FUNCTION_BLOCK FB_Mixer_Ctrl
VAR_INPUT
	i_Interlocks		:ARRAY[1..5] OF BOOL;
	i_AutoCmdFwd		:BOOL;
	i_AutoCmdBcw		:BOOL;
	i_AutoSpeedSP		:REAL;
	i_ManCmdFwd			:BOOL;
	i_ManCmdBcw			:BOOL;
	i_ManStop			:BOOL;
	i_ManSpeedSP		:REAL;
	i_SpeedAP			:REAL;
	i_CurrentAP			:REAL;
	i_ServiceMode		:BOOL;
END_VAR
VAR_OUTPUT
	q_InterlocksOK		:BOOL;
	q_bCmdFwd			:BOOL;
	q_bCmdBcw			:BOOL;
	q_rSpeedSP			:REAL;
END_VAR
VAR
	bCmdFwd				:BOOL;
	bCmdBcw				:BOOL;
	tofCMDFwd			:TOF;
	tofCMDBcw			:TOF;
	tonFwdOff			:TON;
	tonBcwOff			:TON;
END_VAR
VAR // added by the converter: edge detectors and wires of the graphical bodies
    _w1 : BOOL;
END_VAR

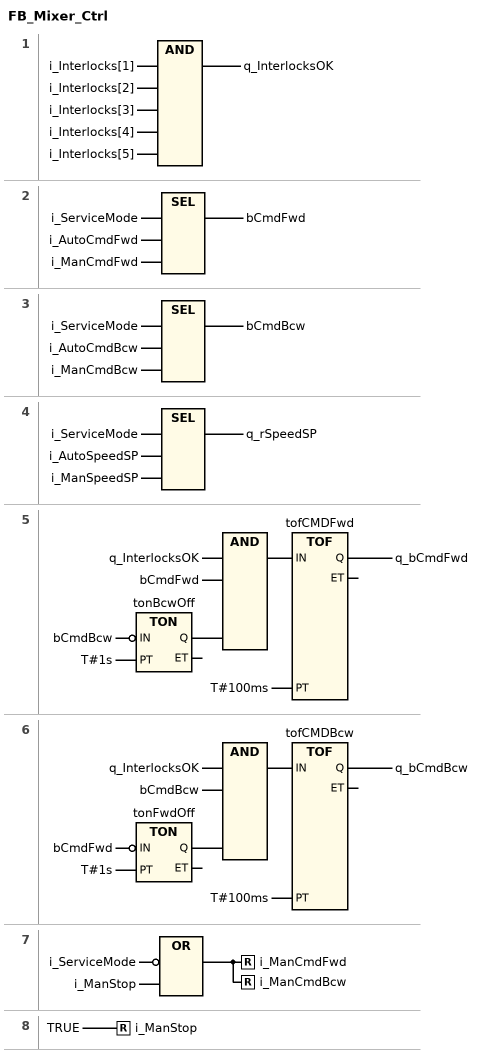
// NETWORK 1
q_InterlocksOK := i_Interlocks[1] AND i_Interlocks[2] AND i_Interlocks[3] AND i_Interlocks[4] AND i_Interlocks[5];

// NETWORK 2
bCmdFwd := SEL(i_ServiceMode, i_AutoCmdFwd, i_ManCmdFwd);

// NETWORK 3
bCmdBcw := SEL(i_ServiceMode, i_AutoCmdBcw, i_ManCmdBcw);

// NETWORK 4
q_rSpeedSP := SEL(i_ServiceMode, i_AutoSpeedSP, i_ManSpeedSP);

// NETWORK 5
tonBcwOff(IN := NOT bCmdBcw, PT := T#1s); // TON
tofCMDFwd(IN := q_InterlocksOK AND bCmdFwd AND tonBcwOff.Q, PT := T#100ms); // TOF
q_bCmdFwd := tofCMDFwd.Q;

// NETWORK 6
tonFwdOff(IN := NOT bCmdFwd, PT := T#1s); // TON
tofCMDBcw(IN := q_InterlocksOK AND bCmdBcw AND tonFwdOff.Q, PT := T#100ms); // TOF
q_bCmdBcw := tofCMDBcw.Q;

// NETWORK 7
_w1 := NOT i_ServiceMode OR i_ManStop;
i_ManCmdFwd R= _w1;
i_ManCmdBcw R= _w1;

// NETWORK 8
i_ManStop R= TRUE;

END_FUNCTION_BLOCK

(* stored: Version 1.1.0.1, ProductVersion 3.1.4024.12
   POU FB_Mixer_Ctrl: Id {49f12b5b-7b3f-4962-9afb-5c64de07ca75}, SpecialFunc None *)
